// TIA Portal V18 export
DATA_BLOCK "Planta_DB"   // DB2
// stored: InstanceOfName Planta, InstanceOfType FB
"Planta"
   // VAR_INPUT
   //    Valve : Bool;
   //    PID_output : Real;
   // END_VAR
   // VAR_OUTPUT
   //    Physvar : Real;
   // END_VAR
   // VAR
   //    F1 : Bool;
   //    F2 : Bool;
   //    F3 : Bool;
   //    F4 : Bool;
   //    F5 : Bool;
   //    F6 : Bool;
   //    LL : Real;
   //    L : Real;
   //    H : Real;
   //    HH : Real;
   //    LL_M : Real;
   //    L_M : Real;
   //    H_M : Real;
   //    HH_M : Real;
   //    MAX_M : Real;
   //    Out_M : Real;
   // END_VAR
BEGIN
END_DATA_BLOCK
